// TIA Portal V15 export
// export: Created 2019-02-11T16:59:47.5610163Z, ExportSetting WithDefaults, WithReadOnly, DisplayName Totally Integrated Automation Portal, DisplayVersion V15 Update 2, DisplayName TIA Portal Openness, DisplayVersion V15 Update 2, DisplayName STEP 7 Professional, DisplayVersion V15 Update 2, DisplayName STEP 7 Safety, DisplayVersion V15, DisplayName WinCC Professional, DisplayVersion V15 Update 2, DisplayName SIMATIC Visualization Architect, DisplayVersion V15 Update 1
DATA_BLOCK "FGDB_FIXTURENAME"   // DB52
TITLE = Geostation
{ S7_Optimized_Access := 'FALSE' }
AUTHOR : integra
FAMILY : SUB
VERSION : 1.0
// stored: AutoNumber true, CodeModifiedDate 2019-02-11T16:59:25.3394383Z, CompileDate 2019-02-11T16:59:38.6723931Z, CreationDate 2019-02-11T16:57:16.7579906Z, DBAccessibleFromOPCUA true, InstanceOfName iFG_PART_LINKING, InstanceOfNumber 4, InstanceOfType FB, InterfaceModifiedDate 2018-02-20T17:35:28.4288607Z, IsConsistent true, IsKnowHowProtected false, ModifiedDate 2019-02-11T16:59:25.3394383Z, ParameterModified 2017-08-28T13:41:12.6207841Z, StructureModified 2018-02-20T16:45:51.3385902Z, UDAEnableTagReadback false
"iFG_PART_LINKING"
   // VAR_INPUT
   //    linkParts : Bool;
   //    partNumber_1 : String[12];
   //    partIdent_1 : String[24];
   //    partNumber_2 { ExternalVisible := 'False'} : String[12];
   //    partIdent_2 : String[24];
   //    partNumber_3 : String[12];
   //    partIdent_3 : String[24];
   //    partNumber_4 : String[12];
   //    partIdent_4 : String[24];
   //    partNumber_5 : String[12];
   //    partIdent_5 : String[24];
   //    partNumber_6 : String[12];
   //    partIdent_6 : String[24];
   //    partNumber_7 : String[12];
   //    partIdent_7 : String[24];
   //    partNumber_8 : String[12];
   //    partIdent_8 : String[24];
   //    partNumber_9 : String[12];
   //    partIdent_9 : String[24];
   //    partNumber_10 : String[12];
   //    partIdent_10 : String[24];
   //    productNumber : String[12];
   //    productIdent : String[24];
   // END_VAR
   // VAR_OUTPUT
   //    fault : Bool;
   //    faultExt : Bool;
   // END_VAR
   // VAR_IN_OUT
   //    RingBuffer : "iUDT_FG_PART_LINKING_RING_BUFFER";
   // END_VAR
   // VAR RETAIN
   //    idx : Int;
   //    sectionNumber : Int;
   //    deskNumber : Int;
   //    stationNumber : Int;
   //    dbNumber : Int;
   //    function : Int;
   //    numberInternalMessages : Int;
   //    numberExternalMessages : Int;
   //    Settings : Struct
   //       PartNumbers : Array[1..20] of String[12];
   //    END_STRUCT;
   //    IfcFGExternal : "iUDT_IFC_SYS_EXTERNAL_ALARM";
   //    ExtP : Struct
   //       setup : Bool;
   //       auto : Bool;
   //       enableIn : Bool;
   //       ack : Bool;
   //    END_STRUCT;
   //    StM : Struct
   //       fault : Bool;
   //       setup : Bool;
   //       auto : Bool;
   //       warning : Bool;
   //       eStop : Bool;
   //       safetyStop : Bool;
   //       enableIn : Bool;
   //       enableOutForward : Bool;
   //       enableOutBackward : Bool;
   //       faultPr : Bool;
   //       pairMon : Bool;
   //       specialMode : Bool;
   //       "13" : Bool;
   //       "14" : Bool;
   //       "15" : Bool;
   //       "16" : Bool;
   //       "17" : Bool;
   //       "18" : Bool;
   //       "19" : Bool;
   //       "20" : Bool;
   //       "21" : Bool;
   //       "22" : Bool;
   //       "23" : Bool;
   //       "24" : Bool;
   //       "25" : Bool;
   //       "26" : Bool;
   //       "27" : Bool;
   //       "28" : Bool;
   //       "29" : Bool;
   //       "30" : Bool;
   //       "31" : Bool;
   //       "32" : Bool;
   //    END_STRUCT;
   //    VB : Struct
   //       "1" : Bool;
   //       "2" : Bool;
   //       "3" : Bool;
   //       "4" : Bool;
   //       "5" : Bool;
   //       "6" : Bool;
   //       "7" : Bool;
   //       "8" : Bool;
   //       "9" : Bool;
   //       "10" : Bool;
   //       "11" : Bool;
   //       "12" : Bool;
   //       "13" : Bool;
   //       "14" : Bool;
   //       "15" : Bool;
   //       "16" : Bool;
   //       "17" : Bool;
   //       "18" : Bool;
   //       "19" : Bool;
   //       "20" : Bool;
   //       "21" : Bool;
   //       "22" : Bool;
   //       "23" : Bool;
   //       "24" : Bool;
   //       "25" : Bool;
   //       "26" : Bool;
   //       "27" : Bool;
   //       "28" : Bool;
   //       "29" : Bool;
   //       "30" : Bool;
   //       "31" : Bool;
   //       "32" : Bool;
   //    END_STRUCT;
   //    VCB : Struct
   //       ack : Bool;
   //    END_STRUCT;
   //    D : Struct
   //       visuAck : Bool;
   //       enableln : Bool;
   //       fPLinkParts : Bool;
   //       newDataSet : Bool;
   //    END_STRUCT;
   //    V : Struct
   //       runtime : UInt;
   //    END_STRUCT;
   // END_VAR
BEGIN
END_DATA_BLOCK
